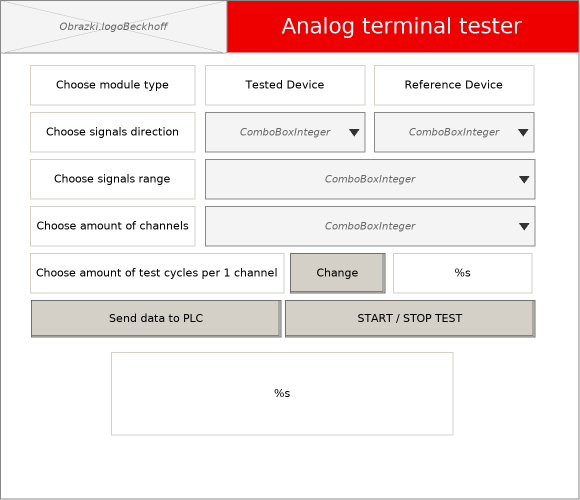
VISUALIZATION Screen1  // 580x500
    Rectangle (225,0 354x52), "Analog terminal tester"
    Image (0,0 227x53), image: Obrazki.logoBeckhoff
    Textfield (30,65 165x40), "Choose module type"
    Textfield (30,253 254x40), "Choose amount of test cycles per 1 channel"
    Button (285,300 250x37), "START / STOP TEST", colour toggle: P_Test.bTestBusy, pressed state: P_Test.bTestBusy
        p573394764: 16#FFFFFF00
        toggle P_Test.bTestEnable
    Button (31,300 250x37), "Send data to PLC", text variable: P_Test.bReadData, colour toggle: P_Test.bErrorReadData
        p573394764: 16#FFFF0000
        tap P_Test.bReadData
    Textfield (30,112 165x40), "Choose signals direction"
    Textfield (30,159 165x40), "Choose signals range"
    Textfield (393,253 139x40), "%s", text variable: P_Test.usiTestCycle
    Textfield (30,206 165x40), "Choose amount of channels"
    Button (290,253 95x40), "Change"
        OnMouseClick: write P_Test.usiTestCycle via VisuDialogs.Numpad, min 1, max 255
    ComboBoxInteger (205,112 160x40), variable: P_Test.eDirection1, text list: 'TL_Direction'
    ComboBoxInteger (205,159 330x40), variable: P_Test.eACtype, text list: 'TL_ACtype'
    ComboBoxInteger (205,206 330x40), variable: P_Test.eNchannel, text list: 'TL_Nchannel'
    Textfield (205,65 160x40), "Tested Device"
    ComboBoxInteger (374,112 160x40), variable: P_Test.eDirection2, text list: 'TL_Direction'
    Textfield (374,65 160x40), "Reference Device"
    Textfield (111,352 342x83), "%s", text variable: P_Test.sStatusBox
END_VISUALIZATION

(* stored: Version 1.1.0.1, ProductVersion 3.1.4020.3
   Visu Screen1: Id {ed43a100-04a8-4dac-a230-1b97ba00f71c} *)
